TYPE ST_STRUCT :
STRUCT
	bVar  : BOOL;
	dtVar : DT;
	fVar  : LREAL;
END_STRUCT
END_TYPE

(* stored: Version 1.1.0.1
   DUT ST_STRUCT: Id {0cb4bfeb-1a42-42f0-a535-45fba0731062} *)
